{attribute 'qualified_only'}
{attribute 'strict'}
TYPE E_ScaleCmd :
(
	ScaleCmd_None, 
	ScaleCmd_SI, 
	ScaleCmd_S, 
	ScaleCmd_T, 
	ScaleCmd_TA, 
	ScaleCmd_TAC
);
END_TYPE

(* stored: Version 1.1.0.1, ProductVersion 3.1.4024.12
   DUT E_ScaleCmd: Id {bb6e26fb-ae72-474f-af7d-1d233df97465} *)
